Staubli VAL3: gestureSpread.pgx

program gestureSpread()
begin
  //open(tClaw)
end
